FUNCTION BYTE_TO_ST08B
  (* Standard: 61499-1 *)
  (* Version 1.0, 2024-02-22, franz *)
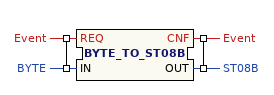
  EVENT_INPUT
    REQ WITH IN; (* Normal Execution Request *)
  END_EVENT
  EVENT_OUTPUT
    CNF WITH OUT; (* Execution Confirmation *)
  END_EVENT
  VAR_INPUT
    IN : BYTE; (* BYTE Input *)
  END_VAR
  VAR_OUTPUT
    OUT : ST08B; (* ST08B Output *)
  END_VAR
  BODY IN ST:
FUNCTION BYTE_TO_ST08B

VAR_INPUT
	IN : BYTE;    // BYTE Input
END_VAR

VAR_OUTPUT
	OUT : ST08B;    // ST08B Output
END_VAR

(* this Function extracts the 8 BOOLS from a byte *)
OUT.B_00 := IN.0;
OUT.B_01 := IN.1;
OUT.B_02 := IN.2;
OUT.B_03 := IN.3;
OUT.B_04 := IN.4;
OUT.B_05 := IN.5;
OUT.B_06 := IN.6;
OUT.B_07 := IN.7;

END_FUNCTION
  END_BODY
END_FUNCTION
